PROGRAM single
VAR
	axisx: AXIS_REF;

	mcPower: MC_Power;
	shouldPowerOn: BOOL;
	isMotorReady: BOOL;
	
	mcSetPosition: MC_SetPosition;
	shouldSetZero: BOOL;
	
	mcJog: MC_Jog;
	shouldJog: BOOL;
	jogDirection: BOOL;
	
	mcMoveRelative: MC_MoveRelative;
	shouldMoveRel: BOOL;
	
	mcHalt: MC_Halt;
	shouldHalt: BOOL;
	
	mcStop: MC_Stop;
	shouldStop:BOOL;
	
	mcReset: MC_Reset;
	shouldReset: BOOL;
	
	mcMoveVelocity: MC_MoveVelocity;
	shouldAdjustVelocity: BOOL;
	velocity: INT;
	
	mcHome: MC_Home;
	shouldGoHome: BOOL;
	homeTrigger: BOOL;
END_VAR

METHOD checkAdjustingVelocity : BOOL
VAR
END_VAR
IF isMotorReady THEN
	mcMoveVelocity(
		Axis:= axisx, 
		Execute:= shouldAdjustVelocity,
		Velocity:= velocity );
END_IF
END_METHOD

METHOD checkGoHome : BOOL
VAR_INPUT
END_VAR
mcHome(
	Axis:= axisx, 
	Execute:= shouldGoHome, 
	Position:= 0, 
	bCalibrationCam:= homeTrigger
);
END_METHOD

METHOD checkHalt : BOOL
VAR_INPUT
END_VAR
IF isMotorReady THEN
	mcHalt(
		Axis:= axisx, 
		Execute:= shouldHalt);
END_IF
END_METHOD

METHOD checkMoving : BOOL
VAR_STAT
END_VAR
IF isMotorReady THEN
	IF shouldJog THEN
		IF jogDirection THEN
		mcJog(
			Axis:= axisx, 
			JogForward:= TRUE, 
			JogBackwards:= FALSE,
			Velocity:= 50);
		ELSE
			mcJog(
				Axis:= axisx, 
				JogForward:= FALSE, 
				JogBackwards:= TRUE,
				Velocity:= 50);
		END_IF
	END_IF
END_IF
END_METHOD

METHOD checkPower : BOOL
VAR_INPUT
END_VAR
VAR
END_VAR
mcPower(
	Axis:= axisx, 
	Enable:= shouldPowerOn, 
	Enable_Positive:= TRUE, 
	Enable_Negative:= TRUE,
	Status=> isMotorReady);
END_METHOD

METHOD checkRelMove : BOOL
VAR_STAT
END_VAR
IF isMotorReady THEN
	mcMoveRelative(
		Axis:= axisx, 
		Execute:= shouldMoveRel, 
		Distance:= 2000, 
		Velocity:= 50);
END_IF;
END_METHOD

METHOD checkReset : BOOL
IF isMotorReady THEN
	mcReset(
		Axis:= axisx, 
		Execute:= shouldReset);
END_IF
END_METHOD

ACTION checkSetPoint:
mcSetPosition(
	Axis:= axisx, 
	Execute:= shouldSetZero,
	Position := 0);
END_ACTION

METHOD checkStop : BOOL
VAR

END_VAR
IF isMotorReady THEN
	mcStop(
		Axis:= axisx, 
		Execute:= shouldStop);
END_IF
END_METHOD

END_PROGRAM

(* stored: Version 1.1.0.1, ProductVersion 3.1.4024.4
   POU single: Id {27ad2594-0b06-4e02-974d-b9c25c9ba880}, SpecialFunc None
   Method checkAdjustingVelocity: Id {9e6ce4d7-1e52-4b34-bfb2-72fdd70b046a}
   Method checkGoHome: Id {7375619a-1d8c-4819-9be5-1e8c5db522ae}
   Method checkHalt: Id {2e1dea5c-2b37-4412-9100-9f336f38a53a}
   Method checkMoving: Id {09805a7c-6bc1-4dd6-8c96-108ff965a2e0}
   Method checkPower: Id {c64668b3-b8f3-4c8c-9e2d-b6feb4467932}
   Method checkRelMove: Id {5a093290-3d42-43f3-afd9-4ef4314b7508}
   Method checkReset: Id {524a7df7-b01b-404f-8b9e-670d73e37929}
   Action checkSetPoint: Id {3147e69a-6538-4ecd-b3b7-7219cbda6e48}
   Method checkStop: Id {59d6d916-623b-4e33-a0e3-1cfdd666254e} *)
